(* IEC 61131-3 sources: Summary-ETFA22/ahorn/benchmark/PPU/Scenario2v0_Final, 4 files *)

(* ---- Scenario2v0_Final.st ---- *)
TYPE
    Magazin_states_t : (Green_Lamp , Init , Interstep , Magazin_Init , Magazin_Init_2 , Slider_Move_Back , Start_Magazin , Step0 , Step1 , convey);
    Crane_states_t : (Crane_Init , Crane_Init_2 , Crane_Lift_Conveyor , Crane_On_Conveyor , Crane_On_Conveyor_Metallic , Crane_Stop , Crane_Turn_Left_Metallic , Crane_Turn_Left_NOT_Metallic , Init , Interstep , Interstep_2 , Interstep_Check_Workpiece , Magazin_Stop , Start_Crane , Step0 , TimeDelay , Turn_Right , release);
END_TYPE

FUNCTION_BLOCK Magazin
    VAR_INPUT  CraneDown : BOOL; END_VAR (*Irwxp*)
    VAR_OUTPUT  CraneLower : BOOL; END_VAR (*Orwxp*)
    VAR_INPUT  CraneOnConveyor : BOOL; END_VAR (*Irwxp*)
    VAR_INPUT  CraneOnMagazin : BOOL; END_VAR (*Irwxp*)
    VAR_INPUT  CraneSucked : BOOL; END_VAR (*Irwxp*)
    VAR_OUTPUT  CraneTurnClockwise : BOOL; END_VAR (*Orwxp*)
    VAR_OUTPUT  CraneTurnCounterclockwise : BOOL; END_VAR (*Orwxp*)
    VAR_INPUT  CraneUp : BOOL; END_VAR (*Irwxp*)
    VAR_OUTPUT  MagazinGreenLamp : BOOL; END_VAR (*Orwxp*)
    VAR_OUTPUT  MagazinSlider : BOOL; END_VAR (*Orwxp*)
    VAR_OUTPUT  MagazinVacuumOff : BOOL; END_VAR (*Orwxp*)
    VAR_OUTPUT  MagazinVacuumOn : BOOL; END_VAR (*Orwxp*)
    VAR_OUTPUT  MagazinWhiteLamp : BOOL; END_VAR (*Orwxp*)
    VAR  SFCInit : BOOL; END_VAR (*Lrwxp*)
    VAR_INPUT  SFCReset : BOOL; END_VAR (*Irwxp*)
    VAR_INPUT  SliderMovedOut : BOOL; END_VAR (*Irwxp*)
    VAR_INPUT  SliderNotMovedOut : BOOL; END_VAR (*Irwxp*)
    VAR_INPUT  StartButtonMagazin : BOOL; END_VAR (*Irwxp*)
    VAR_OUTPUT  StartCommandMagazin : BOOL; END_VAR (*Orwxp*)
    VAR_INPUT  StartVar : BOOL; END_VAR (*Irwxp*)
    VAR_INPUT  WorkpieceReady : BOOL; END_VAR (*Irwxp*)
    VAR  State : Magazin_states_t; END_VAR (*Lrwxp*)
    VAR  Transit : BOOL; END_VAR (*Lrwxp*)
    VAR  interconnectMagazinStartCommand : BOOL; END_VAR (*Lrwxp*)

    CASE State OF
        Magazin_states_t#Green_Lamp:
            (* begin(State) *)
            (* begin(onEntry) *)
            Transit := FALSE;
            (* end(onEntry) *)
            (* begin(onActive) *)
            MagazinGreenLamp := TRUE;
            interconnectMagazinStartCommand := FALSE;
            (* end(onActive) *)
            (* begin(transition) *)
            IF TRUE THEN
                Transit := TRUE;
                State := Magazin_states_t#Magazin_Init;
            END_IF;
            (* end(transition) *)
            (* begin(onExit) *)
            (* end(onExit) *)
            (* end(State) *)

        Magazin_states_t#Init:
            (* begin(State) *)
            (* begin(onEntry) *)
            Transit := FALSE;
            (* end(onEntry) *)
            (* begin(onActive) *)
            (* end(onActive) *)
            (* begin(transition) *)
            IF TRUE THEN
                Transit := TRUE;
                State := Magazin_states_t#Start_Magazin;
            END_IF;
            (* end(transition) *)
            (* begin(onExit) *)
            (* end(onExit) *)
            (* end(State) *)

        Magazin_states_t#Interstep:
            (* begin(State) *)
            (* begin(onEntry) *)
            Transit := FALSE;
            (* end(onEntry) *)
            (* begin(onActive) *)
            StartCommandMagazin := TRUE;
            (* end(onActive) *)
            (* begin(transition) *)
            IF StartVar THEN
                Transit := TRUE;
                State := Magazin_states_t#convey;
            END_IF;
            (* end(transition) *)
            (* begin(onExit) *)
            (* end(onExit) *)
            (* end(State) *)

        Magazin_states_t#Magazin_Init:
            (* begin(State) *)
            (* begin(onEntry) *)
            Transit := FALSE;
            (* end(onEntry) *)
            (* begin(onActive) *)
            MagazinSlider := TRUE;
            (* end(onActive) *)
            (* begin(transition) *)
            IF TRUE THEN
                Transit := TRUE;
                State := Magazin_states_t#Magazin_Init_2;
            END_IF;
            (* end(transition) *)
            (* begin(onExit) *)
            (* end(onExit) *)
            (* end(State) *)

        Magazin_states_t#Magazin_Init_2:
            (* begin(State) *)
            (* begin(onEntry) *)
            Transit := FALSE;
            (* end(onEntry) *)
            (* begin(onActive) *)
            MagazinSlider := FALSE;
            (* end(onActive) *)
            (* begin(transition) *)
            IF TRUE THEN
                Transit := TRUE;
                State := Magazin_states_t#Interstep;
            END_IF;
            (* end(transition) *)
            (* begin(onExit) *)
            (* end(onExit) *)
            (* end(State) *)

        Magazin_states_t#Slider_Move_Back:
            (* begin(State) *)
            (* begin(onEntry) *)
            Transit := FALSE;
            (* end(onEntry) *)
            (* begin(onActive) *)
            IF ((SliderMovedOut = TRUE) AND (SliderNotMovedOut = FALSE)) THEN
                MagazinSlider := FALSE;
            END_IF;
            (* end(onActive) *)
            (* begin(transition) *)
            IF CraneUp THEN
                Transit := TRUE;
                State := Magazin_states_t#Step1;
            END_IF;
            (* end(transition) *)
            (* begin(onExit) *)
            (* end(onExit) *)
            (* end(State) *)

        Magazin_states_t#Start_Magazin:
            (* begin(State) *)
            (* begin(onEntry) *)
            Transit := FALSE;
            (* end(onEntry) *)
            (* begin(onActive) *)
            MagazinSlider := FALSE;
            MagazinGreenLamp := FALSE;
            StartVar := FALSE;
            StartCommandMagazin := FALSE;
            IF (StartButtonMagazin = TRUE) THEN
                interconnectMagazinStartCommand := TRUE;
            END_IF;
            (* end(onActive) *)
            (* begin(transition) *)
            IF interconnectMagazinStartCommand THEN
                Transit := TRUE;
                State := Magazin_states_t#Green_Lamp;
            END_IF;
            (* end(transition) *)
            (* begin(onExit) *)
            (* end(onExit) *)
            (* end(State) *)

        Magazin_states_t#Step0:
            (* begin(State) *)
            (* begin(onEntry) *)
            Transit := FALSE;
            (* end(onEntry) *)
            (* begin(onActive) *)
            (* end(onActive) *)
            (* begin(transition) *)
            IF CraneDown THEN
                Transit := TRUE;
                State := Magazin_states_t#Slider_Move_Back;
            END_IF;
            (* end(transition) *)
            (* begin(onExit) *)
            (* end(onExit) *)
            (* end(State) *)

        Magazin_states_t#Step1:
            (* begin(State) *)
            (* begin(onEntry) *)
            Transit := FALSE;
            (* end(onEntry) *)
            (* begin(onActive) *)
            (* end(onActive) *)
            (* begin(transition) *)
            IF CraneOnConveyor THEN
                Transit := TRUE;
                State := Magazin_states_t#Interstep;
            END_IF;
            (* end(transition) *)
            (* begin(onExit) *)
            (* end(onExit) *)
            (* end(State) *)

        Magazin_states_t#convey:
            (* begin(State) *)
            (* begin(onEntry) *)
            Transit := FALSE;
            (* end(onEntry) *)
            (* begin(onActive) *)
            IF SliderNotMovedOut THEN
                MagazinSlider := TRUE;
            END_IF;
            (* end(onActive) *)
            (* begin(transition) *)
            IF CraneOnMagazin THEN
                Transit := TRUE;
                State := Magazin_states_t#Step0;
            END_IF;
            (* end(transition) *)
            (* begin(onExit) *)
            (* end(onExit) *)
            (* end(State) *)

            END_CASE;
END_FUNCTION_BLOCK

FUNCTION_BLOCK Crane
    VAR_INPUT  CraneDown : BOOL; END_VAR (*Irwxp*)
    VAR_OUTPUT  CraneLower : BOOL; END_VAR (*Orwxp*)
    VAR_INPUT  CraneOnConveyor : BOOL; END_VAR (*Irwxp*)
    VAR_INPUT  CraneOnMagazin : BOOL; END_VAR (*Irwxp*)
    VAR_INPUT  CraneSucked : BOOL; END_VAR (*Irwxp*)
    VAR_OUTPUT  CraneTurnClockwise : BOOL; END_VAR (*Orwxp*)
    VAR_OUTPUT  CraneTurnCounterclockwise : BOOL; END_VAR (*Orwxp*)
    VAR_INPUT  CraneUp : BOOL; END_VAR (*Irwxp*)
    VAR_INPUT  MagazinCapacitiveSensor : BOOL; END_VAR (*Irwxp*)
    VAR_OUTPUT  MagazinVacuumOff : BOOL; END_VAR (*Orwxp*)
    VAR_OUTPUT  MagazinVacuumOn : BOOL; END_VAR (*Orwxp*)
    VAR  SFCInit : BOOL; END_VAR (*Lrwxp*)
    VAR_INPUT  SFCReset : BOOL; END_VAR (*Irwxp*)
    VAR_INPUT  SliderMovedOut : BOOL; END_VAR (*Irwxp*)
    VAR_INPUT  SliderNotMovedOut : BOOL; END_VAR (*Irwxp*)
    VAR_INPUT  StartButtonMagazin : BOOL; END_VAR (*Irwxp*)
    VAR_OUTPUT  StartCommandCrane : BOOL; END_VAR (*Orwxp*)
    VAR_INPUT  StartVar : BOOL; END_VAR (*Irwxp*)
    VAR  TimeDelay_Timer : TON; END_VAR (*Lrwxp*)
    VAR  TimeDelay_Timer_Duration : TIME := TIME#50.0ms; END_VAR (*Lrwxp*)
    VAR  TimeDelay_Timer_interconnect : BOOL; END_VAR (*Lrwxp*)
    VAR_INPUT  WorkpieceReady : BOOL; END_VAR (*Irwxp*)
    VAR  State : Crane_states_t; END_VAR (*Lrwxp*)
    VAR  Transit : BOOL; END_VAR (*Lrwxp*)
    VAR  interconnectCraneStartCommand : BOOL; END_VAR (*Lrwxp*)

    CASE State OF
        Crane_states_t#Crane_Init:
            (* begin(State) *)
            (* begin(onEntry) *)
            Transit := FALSE;
            (* end(onEntry) *)
            (* begin(onActive) *)
            CraneLower := TRUE;
            interconnectCraneStartCommand := FALSE;
            (* end(onActive) *)
            (* begin(transition) *)
            IF CraneDown THEN
                Transit := TRUE;
                State := Crane_states_t#Crane_Init_2;
            END_IF;
            (* end(transition) *)
            (* begin(onExit) *)
            (* end(onExit) *)
            (* end(State) *)

        Crane_states_t#Crane_Init_2:
            (* begin(State) *)
            (* begin(onEntry) *)
            Transit := FALSE;
            (* end(onEntry) *)
            (* begin(onActive) *)
            CraneLower := FALSE;
            (* end(onActive) *)
            (* begin(transition) *)
            IF CraneUp THEN
                Transit := TRUE;
                State := Crane_states_t#Interstep;
            END_IF;
            (* end(transition) *)
            (* begin(onExit) *)
            (* end(onExit) *)
            (* end(State) *)

        Crane_states_t#Crane_Lift_Conveyor:
            (* begin(State) *)
            (* begin(onEntry) *)
            Transit := FALSE;
            (* end(onEntry) *)
            (* begin(onActive) *)
            CraneLower := FALSE;
            (* end(onActive) *)
            (* begin(transition) *)
            IF TRUE THEN
                Transit := TRUE;
                State := Crane_states_t#Interstep;
            END_IF;
            (* end(transition) *)
            (* begin(onExit) *)
            (* end(onExit) *)
            (* end(State) *)

        Crane_states_t#Crane_On_Conveyor:
            (* begin(State) *)
            (* begin(onEntry) *)
            Transit := FALSE;
            (* end(onEntry) *)
            (* begin(onActive) *)
            CraneTurnCounterclockwise := FALSE;
            CraneTurnClockwise := FALSE;
            CraneLower := TRUE;
            (* end(onActive) *)
            (* begin(transition) *)
            IF CraneDown THEN
                Transit := TRUE;
                State := Crane_states_t#release;
            END_IF;
            (* end(transition) *)
            (* begin(onExit) *)
            (* end(onExit) *)
            (* end(State) *)

        Crane_states_t#Crane_On_Conveyor_Metallic:
            (* begin(State) *)
            (* begin(onEntry) *)
            Transit := FALSE;
            (* end(onEntry) *)
            (* begin(onActive) *)
            CraneTurnCounterclockwise := FALSE;
            CraneTurnClockwise := FALSE;
            CraneLower := TRUE;
            (* end(onActive) *)
            (* begin(transition) *)
            IF CraneDown THEN
                Transit := TRUE;
                State := Crane_states_t#release;
            END_IF;
            (* end(transition) *)
            (* begin(onExit) *)
            (* end(onExit) *)
            (* end(State) *)

        Crane_states_t#Crane_Stop:
            (* begin(State) *)
            (* begin(onEntry) *)
            Transit := FALSE;
            (* end(onEntry) *)
            (* begin(onActive) *)
            (* end(onActive) *)
            (* begin(transition) *)
            IF TRUE THEN
                Transit := TRUE;
                State := Crane_states_t#Start_Crane;
            END_IF;
            (* end(transition) *)
            (* begin(onExit) *)
            (* end(onExit) *)
            (* end(State) *)

        Crane_states_t#Crane_Turn_Left_Metallic:
            (* begin(State) *)
            (* begin(onEntry) *)
            Transit := FALSE;
            (* end(onEntry) *)
            (* begin(onActive) *)
            CraneTurnCounterclockwise := TRUE;
            CraneTurnClockwise := FALSE;
            (* end(onActive) *)
            (* begin(transition) *)
            IF CraneOnConveyor THEN
                Transit := TRUE;
                State := Crane_states_t#Crane_On_Conveyor_Metallic;
            END_IF;
            (* end(transition) *)
            (* begin(onExit) *)
            (* end(onExit) *)
            (* end(State) *)

        Crane_states_t#Crane_Turn_Left_NOT_Metallic:
            (* begin(State) *)
            (* begin(onEntry) *)
            Transit := FALSE;
            (* end(onEntry) *)
            (* begin(onActive) *)
            CraneTurnCounterclockwise := TRUE;
            CraneTurnClockwise := FALSE;
            (* end(onActive) *)
            (* begin(transition) *)
            IF CraneOnConveyor THEN
                Transit := TRUE;
                State := Crane_states_t#Crane_On_Conveyor;
            END_IF;
            (* end(transition) *)
            (* begin(onExit) *)
            (* end(onExit) *)
            (* end(State) *)

        Crane_states_t#Init:
            (* begin(State) *)
            (* begin(onEntry) *)
            Transit := FALSE;
            (* end(onEntry) *)
            (* begin(onActive) *)
            (* end(onActive) *)
            (* begin(transition) *)
            IF TRUE THEN
                Transit := TRUE;
                State := Crane_states_t#Start_Crane;
            END_IF;
            (* end(transition) *)
            (* begin(onExit) *)
            (* end(onExit) *)
            (* end(State) *)

        Crane_states_t#Interstep:
            (* begin(State) *)
            (* begin(onEntry) *)
            Transit := FALSE;
            (* end(onEntry) *)
            (* begin(onActive) *)
            StartCommandCrane := TRUE;
            (* end(onActive) *)
            (* begin(transition) *)
            IF StartVar THEN
                Transit := TRUE;
                State := Crane_states_t#Interstep_2;
            END_IF;
            (* end(transition) *)
            (* begin(onExit) *)
            (* end(onExit) *)
            (* end(State) *)

        Crane_states_t#Interstep_2:
            (* begin(State) *)
            (* begin(onEntry) *)
            Transit := FALSE;
            (* end(onEntry) *)
            (* begin(onActive) *)
            (* end(onActive) *)
            (* begin(transition) *)
            IF SliderMovedOut THEN
                Transit := TRUE;
                State := Crane_states_t#TimeDelay;
            END_IF;
            (* end(transition) *)
            (* begin(onExit) *)
            (* end(onExit) *)
            (* end(State) *)

        Crane_states_t#Interstep_Check_Workpiece:
            (* begin(State) *)
            (* begin(onEntry) *)
            Transit := FALSE;
            (* end(onEntry) *)
            (* begin(onActive) *)
            (* end(onActive) *)
            (* begin(transition) *)
            IF WorkpieceReady THEN
                Transit := TRUE;
                State := Crane_states_t#Magazin_Stop;
            ELSIF NOT WorkpieceReady THEN
                Transit := TRUE;
                State := Crane_states_t#Crane_Stop;
            END_IF;
            (* end(transition) *)
            (* begin(onExit) *)
            (* end(onExit) *)
            (* end(State) *)

        Crane_states_t#Magazin_Stop:
            (* begin(State) *)
            (* begin(onEntry) *)
            Transit := FALSE;
            (* end(onEntry) *)
            (* begin(onActive) *)
            CraneTurnClockwise := FALSE;
            CraneTurnCounterclockwise := FALSE;
            MagazinVacuumOn := TRUE;
            MagazinVacuumOff := FALSE;
            CraneLower := TRUE;
            (* end(onActive) *)
            (* begin(transition) *)
            IF CraneSucked THEN
                Transit := TRUE;
                State := Crane_states_t#Step0;
            END_IF;
            (* end(transition) *)
            (* begin(onExit) *)
            (* end(onExit) *)
            (* end(State) *)

        Crane_states_t#Start_Crane:
            (* begin(State) *)
            (* begin(onEntry) *)
            Transit := FALSE;
            (* end(onEntry) *)
            (* begin(onActive) *)
            CraneLower := FALSE;
            MagazinVacuumOff := TRUE;
            MagazinVacuumOn := FALSE;
            CraneTurnCounterclockwise := FALSE;
            CraneTurnClockwise := FALSE;
            StartVar := FALSE;
            StartCommandCrane := FALSE;
            IF (StartButtonMagazin = TRUE) THEN
                interconnectCraneStartCommand := TRUE;
            END_IF;
            (* end(onActive) *)
            (* begin(transition) *)
            IF interconnectCraneStartCommand THEN
                Transit := TRUE;
                State := Crane_states_t#Crane_Init;
            END_IF;
            (* end(transition) *)
            (* begin(onExit) *)
            (* end(onExit) *)
            (* end(State) *)

        Crane_states_t#Step0:
            (* begin(State) *)
            (* begin(onEntry) *)
            Transit := FALSE;
            (* end(onEntry) *)
            (* begin(onActive) *)
            CraneLower := FALSE;
            (* end(onActive) *)
            (* begin(transition) *)
            IF (CraneUp AND MagazinCapacitiveSensor) THEN
                Transit := TRUE;
                State := Crane_states_t#Crane_Turn_Left_Metallic;
            ELSIF (CraneUp AND NOT MagazinCapacitiveSensor) THEN
                Transit := TRUE;
                State := Crane_states_t#Crane_Turn_Left_NOT_Metallic;
            END_IF;
            (* end(transition) *)
            (* begin(onExit) *)
            (* end(onExit) *)
            (* end(State) *)

        Crane_states_t#TimeDelay:
            (* begin(State) *)
            (* begin(onEntry) *)
            Transit := FALSE;
            (* end(onEntry) *)
            (* begin(onActive) *)
            TimeDelay_Timer(IN := TRUE, PT := TimeDelay_Timer_Duration);
            TimeDelay_Timer_interconnect := TimeDelay_Timer.Q;
            (* end(onActive) *)
            (* begin(transition) *)
            IF TimeDelay_Timer_interconnect THEN
                Transit := TRUE;
                State := Crane_states_t#Turn_Right;
            END_IF;
            (* end(transition) *)
            (* begin(onExit) *)
            (* end(onExit) *)
            (* end(State) *)

        Crane_states_t#Turn_Right:
            (* begin(State) *)
            (* begin(onEntry) *)
            Transit := FALSE;
            (* end(onEntry) *)
            (* begin(onActive) *)
            CraneTurnClockwise := TRUE;
            CraneTurnCounterclockwise := FALSE;
            (* end(onActive) *)
            (* begin(transition) *)
            IF CraneOnMagazin THEN
                Transit := TRUE;
                State := Crane_states_t#Interstep_Check_Workpiece;
            END_IF;
            (* end(transition) *)
            (* begin(onExit) *)
            (* end(onExit) *)
            (* end(State) *)

        Crane_states_t#release:
            (* begin(State) *)
            (* begin(onEntry) *)
            Transit := FALSE;
            (* end(onEntry) *)
            (* begin(onActive) *)
            MagazinVacuumOff := TRUE;
            MagazinVacuumOn := FALSE;
            (* end(onActive) *)
            (* begin(transition) *)
            IF TRUE THEN
                Transit := TRUE;
                State := Crane_states_t#Crane_Lift_Conveyor;
            END_IF;
            (* end(transition) *)
            (* begin(onExit) *)
            (* end(onExit) *)
            (* end(State) *)

            END_CASE;
END_FUNCTION_BLOCK

PROGRAM Main

VAR  Actuator_CraneLower : BOOL; END_VAR (*Lrwxp*)
VAR  Actuator_CraneTurnClockwise : BOOL; END_VAR (*Lrwxp*)
VAR  Actuator_CraneTurnCounterclockwise : BOOL; END_VAR (*Lrwxp*)
VAR  Actuator_MagazinGreenLamp : BOOL; END_VAR (*Lrwxp*)
VAR  Actuator_MagazinSlider : BOOL; END_VAR (*Lrwxp*)
VAR  Actuator_MagazinVacuumOff : BOOL; END_VAR (*Lrwxp*)
VAR  Actuator_MagazinVacuumOn : BOOL; END_VAR (*Lrwxp*)
VAR  Actuator_MagazinWhiteLamp : BOOL; END_VAR (*Lrwxp*)
VAR  Crane : Crane; END_VAR (*Lrwxp*)
VAR  Mag : Magazin; END_VAR (*Lrwxp*)
VAR  Sensor_CraneDown : BOOL; END_VAR (*Lrwxp*)
VAR  Sensor_CraneOnConveyor : BOOL; END_VAR (*Lrwxp*)
VAR  Sensor_CraneOnMagazin : BOOL; END_VAR (*Lrwxp*)
VAR  Sensor_CranePosition : BOOL; END_VAR (*Lrwxp*)
VAR  Sensor_CranePositionStamp : BOOL; END_VAR (*Lrwxp*)
VAR  Sensor_CraneSucked : BOOL; END_VAR (*Lrwxp*)
VAR  Sensor_CraneUp : BOOL; END_VAR (*Lrwxp*)
VAR  Sensor_MagazinCapacitiveSensor : BOOL; END_VAR (*Lrwxp*)
VAR  Sensor_MagazinEmergencyStop : BOOL; END_VAR (*Lrwxp*)
VAR  Sensor_MagazinOpticalSensor : BOOL; END_VAR (*Lrwxp*)
VAR  Sensor_MagazinSwitchManuellAutomatic : BOOL; END_VAR (*Lrwxp*)
VAR  Sensor_SliderMovedOut : BOOL; END_VAR (*Lrwxp*)
VAR  Sensor_SliderNotMovedOut : BOOL; END_VAR (*Lrwxp*)
VAR  Sensor_StartButtonMagazin : BOOL; END_VAR (*Lrwxp*)
VAR  Sensor_WorkpieceReady : BOOL; END_VAR (*Lrwxp*)
Mag.SliderNotMovedOut := Sensor_SliderNotMovedOut;
Mag.SliderMovedOut := Sensor_SliderMovedOut;
Mag.CraneOnMagazin := Sensor_CraneOnMagazin;
Mag.CraneDown := Sensor_CraneDown;
Mag.CraneUp := Sensor_CraneUp;
Mag.CraneOnConveyor := Sensor_CraneOnConveyor;
Mag.WorkpieceReady := Sensor_WorkpieceReady;
Mag.StartButtonMagazin := Sensor_StartButtonMagazin;
Actuator_MagazinSlider := Mag.MagazinSlider;
Actuator_MagazinGreenLamp := Mag.MagazinGreenLamp;
Crane.WorkpieceReady := Sensor_WorkpieceReady;
Crane.CraneUp := Sensor_CraneUp;
Crane.CraneOnConveyor := Sensor_CraneOnConveyor;
Crane.CraneDown := Sensor_CraneDown;
Crane.CraneSucked := Sensor_CraneSucked;
Crane.CraneOnMagazin := Sensor_CraneOnMagazin;
Crane.MagazinCapacitiveSensor := Sensor_MagazinCapacitiveSensor;
Crane.SliderMovedOut := Sensor_SliderMovedOut;
Crane.StartButtonMagazin := Sensor_StartButtonMagazin;
Actuator_CraneTurnCounterclockwise := Crane.CraneTurnCounterclockwise;
Actuator_CraneTurnClockwise := Crane.CraneTurnClockwise;
Actuator_CraneLower := Crane.CraneLower;
Actuator_MagazinVacuumOff := Crane.MagazinVacuumOff;
Actuator_MagazinVacuumOn := Crane.MagazinVacuumOn;
IF Sensor_MagazinEmergencyStop THEN
    Mag();
    Crane();
    IF Actuator_MagazinGreenLamp THEN
        IF (Crane.StartCommandCrane AND Mag.StartCommandMagazin) THEN
            Crane.StartVar := TRUE;
            Mag.StartVar := TRUE;
        END_IF;
    END_IF;
    Crane.SFCReset := FALSE;
    Mag.SFCReset := FALSE;
ELSIF NOT Sensor_MagazinEmergencyStop THEN
    Actuator_MagazinSlider := FALSE;
    Actuator_CraneLower := FALSE;
    Actuator_MagazinVacuumOn := FALSE;
    Actuator_MagazinVacuumOff := TRUE;
    Actuator_MagazinGreenLamp := FALSE;
    Actuator_CraneTurnCounterclockwise := FALSE;
    Actuator_CraneTurnClockwise := FALSE;
    Crane.SFCReset := TRUE;
    Mag.SFCReset := TRUE;
    Crane.StartVar := FALSE;
    Mag.StartVar := FALSE;
END_IF;
END_PROGRAM

(* ---- Scenario2v0_Final_Crane.st ---- *)
FUNCTION_BLOCK Crane
    VAR_INPUT  CraneDown : BOOL; END_VAR (*Irwxp*)
    VAR_OUTPUT  CraneLower : BOOL; END_VAR (*Orwxp*)
    VAR_INPUT  CraneOnConveyor : BOOL; END_VAR (*Irwxp*)
    VAR_INPUT  CraneOnMagazin : BOOL; END_VAR (*Irwxp*)
    VAR_INPUT  CraneSucked : BOOL; END_VAR (*Irwxp*)
    VAR_OUTPUT  CraneTurnClockwise : BOOL; END_VAR (*Orwxp*)
    VAR_OUTPUT  CraneTurnCounterclockwise : BOOL; END_VAR (*Orwxp*)
    VAR_INPUT  CraneUp : BOOL; END_VAR (*Irwxp*)
    VAR_INPUT  MagazinCapacitiveSensor : BOOL; END_VAR (*Irwxp*)
    VAR_OUTPUT  MagazinVacuumOff : BOOL; END_VAR (*Orwxp*)
    VAR_OUTPUT  MagazinVacuumOn : BOOL; END_VAR (*Orwxp*)
    VAR  SFCInit : BOOL; END_VAR (*Lrwxp*)
    VAR_INPUT  SFCReset : BOOL; END_VAR (*Irwxp*)
    VAR_INPUT  SliderMovedOut : BOOL; END_VAR (*Irwxp*)
    VAR_INPUT  SliderNotMovedOut : BOOL; END_VAR (*Irwxp*)
    VAR_INPUT  StartButtonMagazin : BOOL; END_VAR (*Irwxp*)
    VAR_OUTPUT  StartCommandCrane : BOOL; END_VAR (*Orwxp*)
    VAR_INPUT  StartVar : BOOL; END_VAR (*Irwxp*)
    VAR  TimeDelay_Timer : TON; END_VAR (*Lrwxp*)
    VAR  TimeDelay_Timer_Duration : TIME := TIME#50.0ms; END_VAR (*Lrwxp*)
    VAR  TimeDelay_Timer_interconnect : BOOL; END_VAR (*Lrwxp*)
    VAR_INPUT  WorkpieceReady : BOOL; END_VAR (*Irwxp*)
    VAR  State : Crane_states_t; END_VAR (*Lrwxp*)
    VAR  Transit : BOOL; END_VAR (*Lrwxp*)
    VAR  interconnectCraneStartCommand : BOOL; END_VAR (*Lrwxp*)

    CASE State OF
        Crane_states_t#Crane_Init:
            (* begin(State) *)
            (* begin(onEntry) *)
            Transit := FALSE;
            (* end(onEntry) *)
            (* begin(onActive) *)
            CraneLower := TRUE;
            interconnectCraneStartCommand := FALSE;
            (* end(onActive) *)
            (* begin(transition) *)
            IF CraneDown THEN
                Transit := TRUE;
                State := Crane_states_t#Crane_Init_2;
            END_IF;
            (* end(transition) *)
            (* begin(onExit) *)
            (* end(onExit) *)
            (* end(State) *)

        Crane_states_t#Crane_Init_2:
            (* begin(State) *)
            (* begin(onEntry) *)
            Transit := FALSE;
            (* end(onEntry) *)
            (* begin(onActive) *)
            CraneLower := FALSE;
            (* end(onActive) *)
            (* begin(transition) *)
            IF CraneUp THEN
                Transit := TRUE;
                State := Crane_states_t#Interstep;
            END_IF;
            (* end(transition) *)
            (* begin(onExit) *)
            (* end(onExit) *)
            (* end(State) *)

        Crane_states_t#Crane_Lift_Conveyor:
            (* begin(State) *)
            (* begin(onEntry) *)
            Transit := FALSE;
            (* end(onEntry) *)
            (* begin(onActive) *)
            CraneLower := FALSE;
            (* end(onActive) *)
            (* begin(transition) *)
            IF TRUE THEN
                Transit := TRUE;
                State := Crane_states_t#Interstep;
            END_IF;
            (* end(transition) *)
            (* begin(onExit) *)
            (* end(onExit) *)
            (* end(State) *)

        Crane_states_t#Crane_On_Conveyor:
            (* begin(State) *)
            (* begin(onEntry) *)
            Transit := FALSE;
            (* end(onEntry) *)
            (* begin(onActive) *)
            CraneTurnCounterclockwise := FALSE;
            CraneTurnClockwise := FALSE;
            CraneLower := TRUE;
            (* end(onActive) *)
            (* begin(transition) *)
            IF CraneDown THEN
                Transit := TRUE;
                State := Crane_states_t#release;
            END_IF;
            (* end(transition) *)
            (* begin(onExit) *)
            (* end(onExit) *)
            (* end(State) *)

        Crane_states_t#Crane_On_Conveyor_Metallic:
            (* begin(State) *)
            (* begin(onEntry) *)
            Transit := FALSE;
            (* end(onEntry) *)
            (* begin(onActive) *)
            CraneTurnCounterclockwise := FALSE;
            CraneTurnClockwise := FALSE;
            CraneLower := TRUE;
            (* end(onActive) *)
            (* begin(transition) *)
            IF CraneDown THEN
                Transit := TRUE;
                State := Crane_states_t#release;
            END_IF;
            (* end(transition) *)
            (* begin(onExit) *)
            (* end(onExit) *)
            (* end(State) *)

        Crane_states_t#Crane_Stop:
            (* begin(State) *)
            (* begin(onEntry) *)
            Transit := FALSE;
            (* end(onEntry) *)
            (* begin(onActive) *)
            (* end(onActive) *)
            (* begin(transition) *)
            IF TRUE THEN
                Transit := TRUE;
                State := Crane_states_t#Start_Crane;
            END_IF;
            (* end(transition) *)
            (* begin(onExit) *)
            (* end(onExit) *)
            (* end(State) *)

        Crane_states_t#Crane_Turn_Left_Metallic:
            (* begin(State) *)
            (* begin(onEntry) *)
            Transit := FALSE;
            (* end(onEntry) *)
            (* begin(onActive) *)
            CraneTurnCounterclockwise := TRUE;
            CraneTurnClockwise := FALSE;
            (* end(onActive) *)
            (* begin(transition) *)
            IF CraneOnConveyor THEN
                Transit := TRUE;
                State := Crane_states_t#Crane_On_Conveyor_Metallic;
            END_IF;
            (* end(transition) *)
            (* begin(onExit) *)
            (* end(onExit) *)
            (* end(State) *)

        Crane_states_t#Crane_Turn_Left_NOT_Metallic:
            (* begin(State) *)
            (* begin(onEntry) *)
            Transit := FALSE;
            (* end(onEntry) *)
            (* begin(onActive) *)
            CraneTurnCounterclockwise := TRUE;
            CraneTurnClockwise := FALSE;
            (* end(onActive) *)
            (* begin(transition) *)
            IF CraneOnConveyor THEN
                Transit := TRUE;
                State := Crane_states_t#Crane_On_Conveyor;
            END_IF;
            (* end(transition) *)
            (* begin(onExit) *)
            (* end(onExit) *)
            (* end(State) *)

        Crane_states_t#Init:
            (* begin(State) *)
            (* begin(onEntry) *)
            Transit := FALSE;
            (* end(onEntry) *)
            (* begin(onActive) *)
            (* end(onActive) *)
            (* begin(transition) *)
            IF TRUE THEN
                Transit := TRUE;
                State := Crane_states_t#Start_Crane;
            END_IF;
            (* end(transition) *)
            (* begin(onExit) *)
            (* end(onExit) *)
            (* end(State) *)

        Crane_states_t#Interstep:
            (* begin(State) *)
            (* begin(onEntry) *)
            Transit := FALSE;
            (* end(onEntry) *)
            (* begin(onActive) *)
            StartCommandCrane := TRUE;
            (* end(onActive) *)
            (* begin(transition) *)
            IF StartVar THEN
                Transit := TRUE;
                State := Crane_states_t#Interstep_2;
            END_IF;
            (* end(transition) *)
            (* begin(onExit) *)
            (* end(onExit) *)
            (* end(State) *)

        Crane_states_t#Interstep_2:
            (* begin(State) *)
            (* begin(onEntry) *)
            Transit := FALSE;
            (* end(onEntry) *)
            (* begin(onActive) *)
            (* end(onActive) *)
            (* begin(transition) *)
            IF SliderMovedOut THEN
                Transit := TRUE;
                State := Crane_states_t#TimeDelay;
            END_IF;
            (* end(transition) *)
            (* begin(onExit) *)
            (* end(onExit) *)
            (* end(State) *)

        Crane_states_t#Interstep_Check_Workpiece:
            (* begin(State) *)
            (* begin(onEntry) *)
            Transit := FALSE;
            (* end(onEntry) *)
            (* begin(onActive) *)
            (* end(onActive) *)
            (* begin(transition) *)
            IF WorkpieceReady THEN
                Transit := TRUE;
                State := Crane_states_t#Magazin_Stop;
            ELSIF NOT WorkpieceReady THEN
                Transit := TRUE;
                State := Crane_states_t#Crane_Stop;
            END_IF;
            (* end(transition) *)
            (* begin(onExit) *)
            (* end(onExit) *)
            (* end(State) *)

        Crane_states_t#Magazin_Stop:
            (* begin(State) *)
            (* begin(onEntry) *)
            Transit := FALSE;
            (* end(onEntry) *)
            (* begin(onActive) *)
            CraneTurnClockwise := FALSE;
            CraneTurnCounterclockwise := FALSE;
            MagazinVacuumOn := TRUE;
            MagazinVacuumOff := FALSE;
            CraneLower := TRUE;
            (* end(onActive) *)
            (* begin(transition) *)
            IF CraneSucked THEN
                Transit := TRUE;
                State := Crane_states_t#Step0;
            END_IF;
            (* end(transition) *)
            (* begin(onExit) *)
            (* end(onExit) *)
            (* end(State) *)

        Crane_states_t#Start_Crane:
            (* begin(State) *)
            (* begin(onEntry) *)
            Transit := FALSE;
            (* end(onEntry) *)
            (* begin(onActive) *)
            CraneLower := FALSE;
            MagazinVacuumOff := TRUE;
            MagazinVacuumOn := FALSE;
            CraneTurnCounterclockwise := FALSE;
            CraneTurnClockwise := FALSE;
            StartVar := FALSE;
            StartCommandCrane := FALSE;
            IF (StartButtonMagazin = TRUE) THEN
                interconnectCraneStartCommand := TRUE;
            END_IF;
            (* end(onActive) *)
            (* begin(transition) *)
            IF interconnectCraneStartCommand THEN
                Transit := TRUE;
                State := Crane_states_t#Crane_Init;
            END_IF;
            (* end(transition) *)
            (* begin(onExit) *)
            (* end(onExit) *)
            (* end(State) *)

        Crane_states_t#Step0:
            (* begin(State) *)
            (* begin(onEntry) *)
            Transit := FALSE;
            (* end(onEntry) *)
            (* begin(onActive) *)
            CraneLower := FALSE;
            (* end(onActive) *)
            (* begin(transition) *)
            IF (CraneUp AND MagazinCapacitiveSensor) THEN
                Transit := TRUE;
                State := Crane_states_t#Crane_Turn_Left_Metallic;
            ELSIF (CraneUp AND NOT MagazinCapacitiveSensor) THEN
                Transit := TRUE;
                State := Crane_states_t#Crane_Turn_Left_NOT_Metallic;
            END_IF;
            (* end(transition) *)
            (* begin(onExit) *)
            (* end(onExit) *)
            (* end(State) *)

        Crane_states_t#TimeDelay:
            (* begin(State) *)
            (* begin(onEntry) *)
            Transit := FALSE;
            (* end(onEntry) *)
            (* begin(onActive) *)
            TimeDelay_Timer(IN := TRUE, PT := TimeDelay_Timer_Duration);
            TimeDelay_Timer_interconnect := TimeDelay_Timer.Q;
            (* end(onActive) *)
            (* begin(transition) *)
            IF TimeDelay_Timer_interconnect THEN
                Transit := TRUE;
                State := Crane_states_t#Turn_Right;
            END_IF;
            (* end(transition) *)
            (* begin(onExit) *)
            (* end(onExit) *)
            (* end(State) *)

        Crane_states_t#Turn_Right:
            (* begin(State) *)
            (* begin(onEntry) *)
            Transit := FALSE;
            (* end(onEntry) *)
            (* begin(onActive) *)
            CraneTurnClockwise := TRUE;
            CraneTurnCounterclockwise := FALSE;
            (* end(onActive) *)
            (* begin(transition) *)
            IF CraneOnMagazin THEN
                Transit := TRUE;
                State := Crane_states_t#Interstep_Check_Workpiece;
            END_IF;
            (* end(transition) *)
            (* begin(onExit) *)
            (* end(onExit) *)
            (* end(State) *)

        Crane_states_t#release:
            (* begin(State) *)
            (* begin(onEntry) *)
            Transit := FALSE;
            (* end(onEntry) *)
            (* begin(onActive) *)
            MagazinVacuumOff := TRUE;
            MagazinVacuumOn := FALSE;
            (* end(onActive) *)
            (* begin(transition) *)
            IF TRUE THEN
                Transit := TRUE;
                State := Crane_states_t#Crane_Lift_Conveyor;
            END_IF;
            (* end(transition) *)
            (* begin(onExit) *)
            (* end(onExit) *)
            (* end(State) *)

            END_CASE;
END_FUNCTION_BLOCK

(* ---- Scenario2v0_Final_Magazin.st ---- *)
FUNCTION_BLOCK Magazin
    VAR_INPUT  CraneDown : BOOL; END_VAR (*Irwxp*)
    VAR_OUTPUT  CraneLower : BOOL; END_VAR (*Orwxp*)
    VAR_INPUT  CraneOnConveyor : BOOL; END_VAR (*Irwxp*)
    VAR_INPUT  CraneOnMagazin : BOOL; END_VAR (*Irwxp*)
    VAR_INPUT  CraneSucked : BOOL; END_VAR (*Irwxp*)
    VAR_OUTPUT  CraneTurnClockwise : BOOL; END_VAR (*Orwxp*)
    VAR_OUTPUT  CraneTurnCounterclockwise : BOOL; END_VAR (*Orwxp*)
    VAR_INPUT  CraneUp : BOOL; END_VAR (*Irwxp*)
    VAR_OUTPUT  MagazinGreenLamp : BOOL; END_VAR (*Orwxp*)
    VAR_OUTPUT  MagazinSlider : BOOL; END_VAR (*Orwxp*)
    VAR_OUTPUT  MagazinVacuumOff : BOOL; END_VAR (*Orwxp*)
    VAR_OUTPUT  MagazinVacuumOn : BOOL; END_VAR (*Orwxp*)
    VAR_OUTPUT  MagazinWhiteLamp : BOOL; END_VAR (*Orwxp*)
    VAR  SFCInit : BOOL; END_VAR (*Lrwxp*)
    VAR_INPUT  SFCReset : BOOL; END_VAR (*Irwxp*)
    VAR_INPUT  SliderMovedOut : BOOL; END_VAR (*Irwxp*)
    VAR_INPUT  SliderNotMovedOut : BOOL; END_VAR (*Irwxp*)
    VAR_INPUT  StartButtonMagazin : BOOL; END_VAR (*Irwxp*)
    VAR_OUTPUT  StartCommandMagazin : BOOL; END_VAR (*Orwxp*)
    VAR_INPUT  StartVar : BOOL; END_VAR (*Irwxp*)
    VAR_INPUT  WorkpieceReady : BOOL; END_VAR (*Irwxp*)
    VAR  State : Magazin_states_t; END_VAR (*Lrwxp*)
    VAR  Transit : BOOL; END_VAR (*Lrwxp*)
    VAR  interconnectMagazinStartCommand : BOOL; END_VAR (*Lrwxp*)

    CASE State OF
        Magazin_states_t#Green_Lamp:
            (* begin(State) *)
            (* begin(onEntry) *)
            Transit := FALSE;
            (* end(onEntry) *)
            (* begin(onActive) *)
            MagazinGreenLamp := TRUE;
            interconnectMagazinStartCommand := FALSE;
            (* end(onActive) *)
            (* begin(transition) *)
            IF TRUE THEN
                Transit := TRUE;
                State := Magazin_states_t#Magazin_Init;
            END_IF;
            (* end(transition) *)
            (* begin(onExit) *)
            (* end(onExit) *)
            (* end(State) *)

        Magazin_states_t#Init:
            (* begin(State) *)
            (* begin(onEntry) *)
            Transit := FALSE;
            (* end(onEntry) *)
            (* begin(onActive) *)
            (* end(onActive) *)
            (* begin(transition) *)
            IF TRUE THEN
                Transit := TRUE;
                State := Magazin_states_t#Start_Magazin;
            END_IF;
            (* end(transition) *)
            (* begin(onExit) *)
            (* end(onExit) *)
            (* end(State) *)

        Magazin_states_t#Interstep:
            (* begin(State) *)
            (* begin(onEntry) *)
            Transit := FALSE;
            (* end(onEntry) *)
            (* begin(onActive) *)
            StartCommandMagazin := TRUE;
            (* end(onActive) *)
            (* begin(transition) *)
            IF StartVar THEN
                Transit := TRUE;
                State := Magazin_states_t#convey;
            END_IF;
            (* end(transition) *)
            (* begin(onExit) *)
            (* end(onExit) *)
            (* end(State) *)

        Magazin_states_t#Magazin_Init:
            (* begin(State) *)
            (* begin(onEntry) *)
            Transit := FALSE;
            (* end(onEntry) *)
            (* begin(onActive) *)
            MagazinSlider := TRUE;
            (* end(onActive) *)
            (* begin(transition) *)
            IF TRUE THEN
                Transit := TRUE;
                State := Magazin_states_t#Magazin_Init_2;
            END_IF;
            (* end(transition) *)
            (* begin(onExit) *)
            (* end(onExit) *)
            (* end(State) *)

        Magazin_states_t#Magazin_Init_2:
            (* begin(State) *)
            (* begin(onEntry) *)
            Transit := FALSE;
            (* end(onEntry) *)
            (* begin(onActive) *)
            MagazinSlider := FALSE;
            (* end(onActive) *)
            (* begin(transition) *)
            IF TRUE THEN
                Transit := TRUE;
                State := Magazin_states_t#Interstep;
            END_IF;
            (* end(transition) *)
            (* begin(onExit) *)
            (* end(onExit) *)
            (* end(State) *)

        Magazin_states_t#Slider_Move_Back:
            (* begin(State) *)
            (* begin(onEntry) *)
            Transit := FALSE;
            (* end(onEntry) *)
            (* begin(onActive) *)
            IF ((SliderMovedOut = TRUE) AND (SliderNotMovedOut = FALSE)) THEN
                MagazinSlider := FALSE;
            END_IF;
            (* end(onActive) *)
            (* begin(transition) *)
            IF CraneUp THEN
                Transit := TRUE;
                State := Magazin_states_t#Step1;
            END_IF;
            (* end(transition) *)
            (* begin(onExit) *)
            (* end(onExit) *)
            (* end(State) *)

        Magazin_states_t#Start_Magazin:
            (* begin(State) *)
            (* begin(onEntry) *)
            Transit := FALSE;
            (* end(onEntry) *)
            (* begin(onActive) *)
            MagazinSlider := FALSE;
            MagazinGreenLamp := FALSE;
            StartVar := FALSE;
            StartCommandMagazin := FALSE;
            IF (StartButtonMagazin = TRUE) THEN
                interconnectMagazinStartCommand := TRUE;
            END_IF;
            (* end(onActive) *)
            (* begin(transition) *)
            IF interconnectMagazinStartCommand THEN
                Transit := TRUE;
                State := Magazin_states_t#Green_Lamp;
            END_IF;
            (* end(transition) *)
            (* begin(onExit) *)
            (* end(onExit) *)
            (* end(State) *)

        Magazin_states_t#Step0:
            (* begin(State) *)
            (* begin(onEntry) *)
            Transit := FALSE;
            (* end(onEntry) *)
            (* begin(onActive) *)
            (* end(onActive) *)
            (* begin(transition) *)
            IF CraneDown THEN
                Transit := TRUE;
                State := Magazin_states_t#Slider_Move_Back;
            END_IF;
            (* end(transition) *)
            (* begin(onExit) *)
            (* end(onExit) *)
            (* end(State) *)

        Magazin_states_t#Step1:
            (* begin(State) *)
            (* begin(onEntry) *)
            Transit := FALSE;
            (* end(onEntry) *)
            (* begin(onActive) *)
            (* end(onActive) *)
            (* begin(transition) *)
            IF CraneOnConveyor THEN
                Transit := TRUE;
                State := Magazin_states_t#Interstep;
            END_IF;
            (* end(transition) *)
            (* begin(onExit) *)
            (* end(onExit) *)
            (* end(State) *)

        Magazin_states_t#convey:
            (* begin(State) *)
            (* begin(onEntry) *)
            Transit := FALSE;
            (* end(onEntry) *)
            (* begin(onActive) *)
            IF SliderNotMovedOut THEN
                MagazinSlider := TRUE;
            END_IF;
            (* end(onActive) *)
            (* begin(transition) *)
            IF CraneOnMagazin THEN
                Transit := TRUE;
                State := Magazin_states_t#Step0;
            END_IF;
            (* end(transition) *)
            (* begin(onExit) *)
            (* end(onExit) *)
            (* end(State) *)

            END_CASE;
END_FUNCTION_BLOCK

(* ---- Scenario2v0_Final_Main.st ---- *)
PROGRAM Main

VAR  Actuator_CraneLower : BOOL; END_VAR (*Lrwxp*)
VAR  Actuator_CraneTurnClockwise : BOOL; END_VAR (*Lrwxp*)
VAR  Actuator_CraneTurnCounterclockwise : BOOL; END_VAR (*Lrwxp*)
VAR  Actuator_MagazinGreenLamp : BOOL; END_VAR (*Lrwxp*)
VAR  Actuator_MagazinSlider : BOOL; END_VAR (*Lrwxp*)
VAR  Actuator_MagazinVacuumOff : BOOL; END_VAR (*Lrwxp*)
VAR  Actuator_MagazinVacuumOn : BOOL; END_VAR (*Lrwxp*)
VAR  Actuator_MagazinWhiteLamp : BOOL; END_VAR (*Lrwxp*)
VAR  Crane : Crane; END_VAR (*Lrwxp*)
VAR  Mag : Magazin; END_VAR (*Lrwxp*)
VAR  Sensor_CraneDown : BOOL; END_VAR (*Lrwxp*)
VAR  Sensor_CraneOnConveyor : BOOL; END_VAR (*Lrwxp*)
VAR  Sensor_CraneOnMagazin : BOOL; END_VAR (*Lrwxp*)
VAR  Sensor_CranePosition : BOOL; END_VAR (*Lrwxp*)
VAR  Sensor_CranePositionStamp : BOOL; END_VAR (*Lrwxp*)
VAR  Sensor_CraneSucked : BOOL; END_VAR (*Lrwxp*)
VAR  Sensor_CraneUp : BOOL; END_VAR (*Lrwxp*)
VAR  Sensor_MagazinCapacitiveSensor : BOOL; END_VAR (*Lrwxp*)
VAR  Sensor_MagazinEmergencyStop : BOOL; END_VAR (*Lrwxp*)
VAR  Sensor_MagazinOpticalSensor : BOOL; END_VAR (*Lrwxp*)
VAR  Sensor_MagazinSwitchManuellAutomatic : BOOL; END_VAR (*Lrwxp*)
VAR  Sensor_SliderMovedOut : BOOL; END_VAR (*Lrwxp*)
VAR  Sensor_SliderNotMovedOut : BOOL; END_VAR (*Lrwxp*)
VAR  Sensor_StartButtonMagazin : BOOL; END_VAR (*Lrwxp*)
VAR  Sensor_WorkpieceReady : BOOL; END_VAR (*Lrwxp*)
Mag.SliderNotMovedOut := Sensor_SliderNotMovedOut;
Mag.SliderMovedOut := Sensor_SliderMovedOut;
Mag.CraneOnMagazin := Sensor_CraneOnMagazin;
Mag.CraneDown := Sensor_CraneDown;
Mag.CraneUp := Sensor_CraneUp;
Mag.CraneOnConveyor := Sensor_CraneOnConveyor;
Mag.WorkpieceReady := Sensor_WorkpieceReady;
Mag.StartButtonMagazin := Sensor_StartButtonMagazin;
Actuator_MagazinSlider := Mag.MagazinSlider;
Actuator_MagazinGreenLamp := Mag.MagazinGreenLamp;
Crane.WorkpieceReady := Sensor_WorkpieceReady;
Crane.CraneUp := Sensor_CraneUp;
Crane.CraneOnConveyor := Sensor_CraneOnConveyor;
Crane.CraneDown := Sensor_CraneDown;
Crane.CraneSucked := Sensor_CraneSucked;
Crane.CraneOnMagazin := Sensor_CraneOnMagazin;
Crane.MagazinCapacitiveSensor := Sensor_MagazinCapacitiveSensor;
Crane.SliderMovedOut := Sensor_SliderMovedOut;
Crane.StartButtonMagazin := Sensor_StartButtonMagazin;
Actuator_CraneTurnCounterclockwise := Crane.CraneTurnCounterclockwise;
Actuator_CraneTurnClockwise := Crane.CraneTurnClockwise;
Actuator_CraneLower := Crane.CraneLower;
Actuator_MagazinVacuumOff := Crane.MagazinVacuumOff;
Actuator_MagazinVacuumOn := Crane.MagazinVacuumOn;
IF Sensor_MagazinEmergencyStop THEN
    Mag();
    Crane();
    IF Actuator_MagazinGreenLamp THEN
        IF (Crane.StartCommandCrane AND Mag.StartCommandMagazin) THEN
            Crane.StartVar := TRUE;
            Mag.StartVar := TRUE;
        END_IF;
    END_IF;
    Crane.SFCReset := FALSE;
    Mag.SFCReset := FALSE;
ELSIF NOT Sensor_MagazinEmergencyStop THEN
    Actuator_MagazinSlider := FALSE;
    Actuator_CraneLower := FALSE;
    Actuator_MagazinVacuumOn := FALSE;
    Actuator_MagazinVacuumOff := TRUE;
    Actuator_MagazinGreenLamp := FALSE;
    Actuator_CraneTurnCounterclockwise := FALSE;
    Actuator_CraneTurnClockwise := FALSE;
    Crane.SFCReset := TRUE;
    Mag.SFCReset := TRUE;
    Crane.StartVar := FALSE;
    Mag.StartVar := FALSE;
END_IF;
END_PROGRAM
